# EPICS IOC start-up script: iocsh/ethercatmcLongin.iocsh
ethercatmcCreateAsynParam $(MOTOR_PORT) $(ASYNPARAMNAME)      Int32

dbLoadRecords("ethercatmcLongin.template", "P=$(P), R=$(R), MOTOR_PORT=$(MOTOR_PORT), CHNO=$(CHNO), ASYNPARAMNAME=$(ASYNPARAMNAME), DESC=$(DESC), EGU=$(EGU)")
